// TIA Portal V17 export
// export: Created 2022-07-20T06:59:37.5326047Z, ExportSetting WithDefaults, DisplayName Totally Integrated Automation Portal, DisplayVersion V17, DisplayName TIA Portal Openness, DisplayVersion V17, DisplayName TIA Portal Version Control Interface, DisplayVersion V17, DisplayName SINAMICS Startdrive Advanced, DisplayVersion V17, DisplayName SINAMICS Startdrive G130, G150, S120, S150, SINAMICS MV, S210, DisplayVersion V17, DisplayName SINAMICS Startdrive G110M, G120, G120C, G120D, G120P, G115D, DisplayVersion V17, DisplayName STEP 7 Professional, DisplayVersion V17, DisplayName STEP 7 Safety, DisplayVersion V17, DisplayName WinCC Advanced, DisplayVersion V17
FUNCTION_BLOCK "FB10005_Logs"   // FB10005, LAD
TITLE = FB10005_Logs
{ S7_Optimized_Access := 'TRUE' }
AUTHOR : Anirouddh
FAMILY : 1000x_SYSTEM
VERSION : 1.0
// Release note : 
// 1.0 - Feature developped
// stored: AutoNumber false, IsIECCheckEnabled false, IsRetainMemResEnabled false, MemoryReserve 100, SetENOAutomatically false, UDAEnableTagReadback false
   VAR_INPUT
      NumberOfLoggingBooleans : Int;
      NumberOfLoggingInterger : Int;
      NumberOfLoggingReals : Int;
   END_VAR
   VAR_OUTPUT
      LogGenerationDone : Bool;
      LogBufferResetDone : Bool;
      LogFile : Array[0..1999] of String;
   END_VAR
   VAR_IN_OUT
      Enable : Bool;
      GenerateLogFile : Bool;
      Reset : Bool;
      Array_LoggingBooleans : Array[0..499] of Bool;
      Array_LoggingBooleans_VariableName : Array[0..499] of String;
      Array_LoggingIntegers : Array[0..499] of Int;
      Array_LoggingIntegers_VariableName : Array[0..499] of String;
      Array_LoggingReals : Array[0..499] of Real;
      Array_LoggingReals_VariableName : Array[0..499] of String;
   END_VAR
   VAR
      BufferLog_SecondPart_Full { ExternalAccessible := 'False'; ExternalVisible := 'False'; ExternalWritable := 'False'} : Bool;
      i : Int;
      j : Int;
      k1 : Int;
      k2 : Int;
      shift : Int;
      NumberOfLoggingVariables : Int;
      BufferSize : Int;
      LastEmptyIndex : Int;
      GenerateLogStateDiagram : Int;
      ResetLogBufferStateDiagram : Int;
      NumberOfRecordedElement : Int;
      LogTimeStamp : DTL;
      R_TRIG_Reset : R_TRIG;
      "R_TRIG_Clock0.5Hz" : R_TRIG;
      R_TRIG_GenerateLogFile { S7_SetPoint := 'True'} : R_TRIG;
      R_TRIG_ArrayFull { S7_SetPoint := 'True'} : R_TRIG;
      F_TRIG_Reset : F_TRIG;
      Array_LoggingBooleans_RTRIGS { S7_SetPoint := 'True'} : Array[0..499] of R_TRIG;
      Array_LoggingBooleans_FTRIGS { S7_SetPoint := 'True'} : Array[0..499] of F_TRIG;
      Array_LoggingIntegers_PreviousValues { S7_SetPoint := 'True'} : Array[0..499] of Int;
      Array_LoggingIntegers_Changed { S7_SetPoint := 'True'} : Array[0..499] of R_TRIG;
      Array_LoggingReals_PreviousValues : Array[0..499] of Real;
      Array_LoggingReals_Changed { S7_SetPoint := 'True'} : Array[0..499] of R_TRIG;
      BufferLog_TimeStamp_FirstPart { S7_SetPoint := 'True'} : Array[0..999] of DTL;
      BufferLog_VariableName_FirstPart : Array[0..999] of String;
      BufferLog_PreviousValue_FirstPart : Array[0..999] of String;
      BufferLog_CurrentValue_FirstPart : Array[0..999] of String;
      BufferLog_TimeStamp_SecondPart { S7_SetPoint := 'True'} : Array[0..999] of DTL;
      BufferLog_VariableName_SecondPart : Array[0..999] of String;
      BufferLog_PreviousValue_SecondPart : Array[0..999] of String;
      BufferLog_CurrentValue_SecondPart : Array[0..999] of String;
      BufferLog_EmptyDTL : Array[0..999] of DTL;
      BufferLog_EmptyString : Array[0..999] of String;
   END_VAR
   VAR_TEMP
      DateTimeReturnValue : Int;
   END_VAR
   VAR CONSTANT
      WAIT_FOR_BUFFER_RESET : Int := 0;
      RESETTING_IN_PROGRESS : Int := 10;
      BUFFER_RESET_DONE : Int := 20;
      "===========" : Bool;
      WAIT_FOR_LOG_GENERATION_REQUEST : Int := 0;
      GENERATE_LOG_FIRST_PART : Int := 10;
      GENERATE_LOG_SECOND_PART : Int := 20;
      RESET_BUFFER : Int := 30;
      ENABLE_LOG : Int := 40;
      LOG_GENERATION_DONE : Int := 50;
   END_VAR
BEGIN

REGION Network 1 (SCL): First Scan
   IF "FirstScan" THEN
       #Reset := FALSE;
       #LogGenerationDone := FALSE;
       #LastEmptyIndex := 0;
   END_IF;
END_REGION

REGION Network 2 (SCL): Edge Signals & Timers
   REGION TIMERS
   END_REGION

   REGION EDGE SIGNALS
       #R_TRIG_Reset(CLK := #Reset);
       #F_TRIG_Reset(CLK := #Reset);
       #"R_TRIG_Clock0.5Hz"(CLK := "Clock_0.5Hz");
       #R_TRIG_GenerateLogFile(CLK := #GenerateLogFile);
   END_REGION
END_REGION

REGION Network 3 (SCL): Logs Commands
   #NumberOfLoggingVariables := MAX(IN1 := #NumberOfLoggingBooleans, IN2 := #NumberOfLoggingInterger, IN3 := #NumberOfLoggingReals);
   #BufferSize := 1000;
END_REGION

REGION Network 4 (SCL): Logging Management
   IF #Enable THEN
       FOR #i := 0 TO #NumberOfLoggingVariables - 1 DO
           //Array Full Management
           #BufferLog_SecondPart_Full := TRUE;

           //Variable Change Management
           #Array_LoggingBooleans_RTRIGS[#i](CLK := #Array_LoggingBooleans[#i]);
           #Array_LoggingBooleans_FTRIGS[#i](CLK := #Array_LoggingBooleans[#i]);
           #Array_LoggingIntegers_Changed[#i](CLK := #Array_LoggingIntegers_PreviousValues[#i] <> #Array_LoggingIntegers[#i]);
           #Array_LoggingReals_Changed[#i](CLK := #"R_TRIG_Clock0.5Hz".Q AND #Array_LoggingReals_PreviousValues[#i] <> #Array_LoggingReals[#i]);

           //Time Stamp Management
           IF
               #Array_LoggingBooleans_RTRIGS[#i].Q OR
               #Array_LoggingBooleans_FTRIGS[#i].Q OR
               #Array_LoggingIntegers_Changed[#i].Q OR
               #Array_LoggingReals_Changed[#i].Q
           THEN
               #DateTimeReturnValue := RD_SYS_T(#LogTimeStamp);
           END_IF;

           REGION BOOLEANS LOGGING MANAGEMENT
               IF #Array_LoggingBooleans_RTRIGS[#i].Q OR #Array_LoggingBooleans_FTRIGS[#i].Q THEN
                   //Logging the variable
                   #BufferLog_VariableName_SecondPart[#LastEmptyIndex] := #Array_LoggingBooleans_VariableName[#i];
                   #BufferLog_TimeStamp_SecondPart[#LastEmptyIndex] := #LogTimeStamp;
                   IF #Array_LoggingBooleans_RTRIGS[#i].Q THEN
                       #BufferLog_PreviousValue_SecondPart[#LastEmptyIndex] := 'FALSE';
                       #BufferLog_CurrentValue_SecondPart[#LastEmptyIndex] := 'TRUE';
                   ELSIF #Array_LoggingBooleans_FTRIGS[#i].Q THEN
                       #BufferLog_PreviousValue_SecondPart[#LastEmptyIndex] := 'TRUE';
                       #BufferLog_CurrentValue_SecondPart[#LastEmptyIndex] := 'FALSE';
                   END_IF;

                   //Array Index Management
                   #R_TRIG_ArrayFull(CLK := #LastEmptyIndex = #BufferSize - 1);
                   IF #R_TRIG_ArrayFull.Q AND #BufferLog_SecondPart_Full THEN
                       #BufferLog_TimeStamp_FirstPart := #BufferLog_TimeStamp_SecondPart;
                       #BufferLog_VariableName_FirstPart := #BufferLog_VariableName_SecondPart;
                       #BufferLog_PreviousValue_FirstPart := #BufferLog_PreviousValue_SecondPart;
                       #BufferLog_CurrentValue_FirstPart := #BufferLog_CurrentValue_SecondPart;

                       #BufferLog_TimeStamp_SecondPart := #BufferLog_EmptyDTL;
                       #BufferLog_VariableName_SecondPart := #BufferLog_EmptyString;
                       #BufferLog_PreviousValue_SecondPart := #BufferLog_EmptyString;
                       #BufferLog_CurrentValue_SecondPart := #BufferLog_EmptyString;

                       #BufferLog_SecondPart_Full := FALSE;
                       #LastEmptyIndex := 0;
                   ELSE
                       #LastEmptyIndex += 1;
                   END_IF;
               END_IF;
           END_REGION

           REGION INTEGERS LOGGING MANAGEMENT
               IF #Array_LoggingIntegers_Changed[#i].Q THEN
                   //Logging The Variable
                   #BufferLog_VariableName_SecondPart[#LastEmptyIndex] := #Array_LoggingIntegers_VariableName[#i];
                   #BufferLog_TimeStamp_SecondPart[#LastEmptyIndex] := #LogTimeStamp;
                   #BufferLog_PreviousValue_SecondPart[#LastEmptyIndex] := "FC10019_RealToString"(#Array_LoggingIntegers_PreviousValues[#i]);
                   #BufferLog_CurrentValue_SecondPart[#LastEmptyIndex] := "FC10019_RealToString"(#Array_LoggingIntegers[#i]);

                   //Store The Actual Value
                   #Array_LoggingIntegers_PreviousValues[#i] := #Array_LoggingIntegers[#i];

                   //Array Index Management
                   #R_TRIG_ArrayFull(CLK := #LastEmptyIndex = #BufferSize - 1);
                   IF #R_TRIG_ArrayFull.Q AND #BufferLog_SecondPart_Full THEN
                       #BufferLog_TimeStamp_FirstPart := #BufferLog_TimeStamp_SecondPart;
                       #BufferLog_VariableName_FirstPart := #BufferLog_VariableName_SecondPart;
                       #BufferLog_PreviousValue_FirstPart := #BufferLog_PreviousValue_SecondPart;
                       #BufferLog_CurrentValue_FirstPart := #BufferLog_CurrentValue_SecondPart;

                       #BufferLog_TimeStamp_SecondPart := #BufferLog_EmptyDTL;
                       #BufferLog_VariableName_SecondPart := #BufferLog_EmptyString;
                       #BufferLog_PreviousValue_SecondPart := #BufferLog_EmptyString;
                       #BufferLog_CurrentValue_SecondPart := #BufferLog_EmptyString;

                       #BufferLog_SecondPart_Full := FALSE;
                       #LastEmptyIndex := 0;
                   ELSE
                       #LastEmptyIndex += 1;
                   END_IF;
               END_IF;
           END_REGION

           REGION REALS LOGGING MANAGEMENT
               IF #Array_LoggingReals_Changed[#i].Q THEN
                   //Logging The Variable
                   #BufferLog_VariableName_SecondPart[#LastEmptyIndex] := #Array_LoggingReals_VariableName[#i];
                   #BufferLog_TimeStamp_SecondPart[#LastEmptyIndex] := #LogTimeStamp;
                   #BufferLog_PreviousValue_SecondPart[#LastEmptyIndex] := "FC10019_RealToString"(#Array_LoggingReals_PreviousValues[#i]);
                   #BufferLog_CurrentValue_SecondPart[#LastEmptyIndex] := "FC10019_RealToString"(#Array_LoggingReals[#i]);

                   //Store The Actual Value
                   #Array_LoggingReals_PreviousValues[#i] := #Array_LoggingReals[#i];

                   //Array Index Management
                   #R_TRIG_ArrayFull(CLK := #LastEmptyIndex = #BufferSize - 1);
                   IF #R_TRIG_ArrayFull.Q AND #BufferLog_SecondPart_Full THEN
                       #BufferLog_TimeStamp_FirstPart := #BufferLog_TimeStamp_SecondPart;
                       #BufferLog_VariableName_FirstPart := #BufferLog_VariableName_SecondPart;
                       #BufferLog_PreviousValue_FirstPart := #BufferLog_PreviousValue_SecondPart;
                       #BufferLog_CurrentValue_FirstPart := #BufferLog_CurrentValue_SecondPart;

                       #BufferLog_TimeStamp_SecondPart := #BufferLog_EmptyDTL;
                       #BufferLog_VariableName_SecondPart := #BufferLog_EmptyString;
                       #BufferLog_PreviousValue_SecondPart := #BufferLog_EmptyString;
                       #BufferLog_CurrentValue_SecondPart := #BufferLog_EmptyString;

                       #BufferLog_SecondPart_Full := FALSE;
                       #LastEmptyIndex := 0;
                   ELSE
                       #LastEmptyIndex += 1;
                   END_IF;
               END_IF;
           END_REGION
       END_FOR;
   END_IF;
END_REGION

REGION Network 5 (SCL): Reset Management
   CASE #ResetLogBufferStateDiagram OF
       #WAIT_FOR_BUFFER_RESET:
           IF #R_TRIG_Reset.Q THEN
               #LogBufferResetDone := FALSE;
               #ResetLogBufferStateDiagram := #RESETTING_IN_PROGRESS;
           END_IF;
       #RESETTING_IN_PROGRESS:
           //Resetting the Buffer Log
           #BufferLog_VariableName_SecondPart := #BufferLog_EmptyString;
           #BufferLog_TimeStamp_SecondPart := #BufferLog_EmptyDTL;
           #BufferLog_PreviousValue_SecondPart := #BufferLog_EmptyString;
           #BufferLog_CurrentValue_SecondPart := #BufferLog_EmptyString;
           #BufferLog_VariableName_FirstPart := #BufferLog_EmptyString;
           #BufferLog_TimeStamp_FirstPart := #BufferLog_EmptyDTL;
           #BufferLog_PreviousValue_FirstPart := #BufferLog_EmptyString;
           #BufferLog_CurrentValue_FirstPart := #BufferLog_EmptyString;

           //Resetting the index
           #LastEmptyIndex := 0;

           //Condition To Go To Next Step        
           #ResetLogBufferStateDiagram := #BUFFER_RESET_DONE;
       #BUFFER_RESET_DONE:
           #Reset := FALSE;
           #ResetLogBufferStateDiagram := #WAIT_FOR_BUFFER_RESET;
   END_CASE;
END_REGION

REGION Network 6 (SCL): Generate Log File Management
   CASE #GenerateLogStateDiagram OF
       #WAIT_FOR_LOG_GENERATION_REQUEST:
           IF #R_TRIG_GenerateLogFile.Q THEN
               #LogGenerationDone := FALSE;
               #NumberOfRecordedElement := 0;
               #k1 := 0;
               #k2 := 0;
               #Enable := FALSE;
               #Reset := FALSE;
               IF #BufferLog_VariableName_FirstPart[0] = '' THEN
                   #shift := 0;
                   #GenerateLogStateDiagram := #GENERATE_LOG_SECOND_PART;
               ELSE
                   #shift := 1000;
                   #GenerateLogStateDiagram := #GENERATE_LOG_FIRST_PART;
               END_IF;
           END_IF;
       #GENERATE_LOG_FIRST_PART:
           //Log Generation In Progress
           WHILE #k1 <= #NumberOfRecordedElement + 49 DO
               #LogFile[#k1] := CONCAT(IN1 := "FC10018_DateToString"(#BufferLog_TimeStamp_FirstPart[#k2]),
                                       IN2 := ' Variable : ',
                                       IN3 := #BufferLog_VariableName_FirstPart[#k2],
                                       IN4 := ' has changed from ',
                                       IN5 := #BufferLog_PreviousValue_FirstPart[#k2],
                                       IN6 := ' to ',
                                       IN7 := #BufferLog_CurrentValue_FirstPart[#k2]);
               #k1 += 1;
               #k2 += 1;
           END_WHILE;

           //Condition To Go To Next Step
           IF #k1 = 1000 THEN
               #k1 := 0;
               #k2 := 0;
               #NumberOfRecordedElement := 0;
               #GenerateLogStateDiagram := #GENERATE_LOG_SECOND_PART;
           ELSE
               #NumberOfRecordedElement += 50;
               #GenerateLogStateDiagram := #GENERATE_LOG_FIRST_PART;
           END_IF;
       #GENERATE_LOG_SECOND_PART:
           //Log Generation In Progress
           WHILE #k1 <= #NumberOfRecordedElement + 49 DO
               #LogFile[#k1 + #shift] := CONCAT(IN1 := "FC10018_DateToString"(#BufferLog_TimeStamp_SecondPart[#k2]),
                                                IN2 := ' Variable : ',
                                                IN3 := #BufferLog_VariableName_SecondPart[#k2],
                                                IN4 := ' has changed from ',
                                                IN5 := #BufferLog_PreviousValue_SecondPart[#k2],
                                                IN6 := ' to ',
                                                IN7 := #BufferLog_CurrentValue_SecondPart[#k2]);
               #k1 += 1;
               #k2 += 1;
           END_WHILE;

           //Condition To Go To Next Step
           IF #k1 = 1000 THEN
               #LogGenerationDone := TRUE;
               #GenerateLogStateDiagram := #RESET_BUFFER;
           ELSE
               #NumberOfRecordedElement += 50;
               #GenerateLogStateDiagram := #GENERATE_LOG_SECOND_PART;
           END_IF;
       #RESET_BUFFER:
           #Reset := TRUE;
           IF #ResetLogBufferStateDiagram = #BUFFER_RESET_DONE THEN
               #Reset := FALSE;
               #GenerateLogStateDiagram := #ENABLE_LOG;
           END_IF;
       #ENABLE_LOG:
           #Enable := TRUE;
           #Reset := FALSE;
           #GenerateLogStateDiagram := #LOG_GENERATION_DONE;
       #LOG_GENERATION_DONE:
           #GenerateLogStateDiagram := #WAIT_FOR_LOG_GENERATION_REQUEST;
   END_CASE;
END_REGION
END_FUNCTION_BLOCK
